FUNCTION F_RAD2HMS_STRING : STRING
VAR_INPUT
	hh:	LREAL;
END_VAR
VAR
	value:		LREAL;
	hours:		INT;
	minutes:	INT;
	seconds:	LREAL;
	
	sign:	int := 1;
	result:	STRING := '';
	
	fbFormat   : FB_FormatString;
END_VAR

IF hh < 0.0 THEN
	sign	:= -1;
	hh		:= -hh;
END_IF

value := hh / GCL.C_2PI * 24.0; 	// rad to hours


hours	:= TRUNC_INT(value);
minutes := TRUNC_INT((value - hours)*60.0);
seconds := (value - hours - minutes/60.0)*3600.0;

// We the calculation so far the value of 14.999999999 will result
// in 14:59:60.
// We want to correct it to 15:00:00.
IF seconds > 59.999 THEN
	seconds	:= 0.0;
	minutes	:= minutes + 1;
	IF minutes = 60 THEN
		minutes	:= 0;
		hours	:= hours + 1;
	END_IF
// Seconds should never be < 0.0. However, it happens due to rounding
// and the value could be ~ -1.0 e-12.
// Set it to zero in that case.
ELSIF seconds < 0.0 THEN
	seconds := 0.0;
END_IF

hours	:= hours * sign;	// put back the sign

// format a string like "+07:01:02.123"
fbFormat( sFormat  := '%+.2d:%.2d:%06.3f', 
					arg1 := F_INT(hours), 
					arg2 := F_INT(minutes), 
					arg3 := F_LREAL(seconds),
					sOut => result);
					
F_RAD2HMS_STRING	:= result;

END_FUNCTION

(* stored: Version 1.1.0.1, ProductVersion 3.1.4022.16
   POU F_RAD2HMS_STRING: Id {3374b487-8b8e-44cb-908f-fe829b65cc39}, SpecialFunc None *)
